// TIA Portal V15 export
// export: Created 2018-05-30T14:06:14.935436Z, ExportSetting WithDefaults, WithReadOnly, DisplayName Totally Integrated Automation Portal, DisplayVersion V15, DisplayName STEP 7 Professional, DisplayVersion V15, DisplayName WinCC Professional, DisplayVersion V15, DisplayName TIA Portal Openness, DisplayVersion V15
FUNCTION_BLOCK "BST_ANALOG_400"   // FB23, STL
{ S7_Optimized_Access := 'FALSE' }
VERSION : 0.1
// stored: AutoNumber false, CodeModifiedDate 2018-05-30T14:01:37.8315867Z, CompileDate 2018-05-30T14:01:37.8315866Z, CreationDate 2018-05-30T13:57:04.4029473Z, InterfaceModifiedDate 2018-05-30T14:01:33.7723544Z, IsConsistent true, IsKnowHowProtected false, ISMultiInstanceCapable true, IsWriteProtected false, LibraryConformanceStatus The object is library-conformant., ModifiedDate 2018-05-30T14:01:37.8315867Z, ParameterModified 2018-05-30T14:01:33.7723544Z, StructureModified 2018-05-30T14:01:33.7723544Z, UDAEnableTagReadback false
   VAR_INPUT
      wVal : Real;
   END_VAR
   VAR_OUTPUT
      QfVal : Real;
      LIM_Qb01 : Bool;
      LIM_Qb02 : Bool;
      LIM_Qb03 : Bool;
      LIM_b04 : Bool;
      QERR : Bool;
   END_VAR
BEGIN
END_FUNCTION_BLOCK
